// TwinCAT 3 PLC project TcForgeExample
// Title: TcForgeExample
// Company: Home
// ProjectVersion: 2.0.0.0
// ProgramVersion: 3.1.4026.26
// libraries:
//   Tc2_Standard, 3.4.7.0 (Beckhoff Automation GmbH)
//   Tc2_System, 3.10.2.0 (Beckhoff Automation GmbH)
//   Tc3_JsonXml, 3.4.9.0 (Beckhoff Automation GmbH)
//   Tc3_Module, 3.4.7.0 (Beckhoff Automation GmbH)
//   [TcForge], 2.0.0.0 (Home)
// project tree:
//   / PlcTask.TcTTO
//   Assembly/ GVL_HW.TcGVL, MAIN.TcPOU, FB_AssemblyStation.TcPOU, ST_AssemblyInputs.TcDUT, ST_AssemblyOutputs.TcDUT
//   ClampCycle/ FB_ReferenceMachine.TcPOU, E_ReferenceCommand.TcDUT
//   Simulation/ FB_SimulationBridge.TcPOU
//   Actuators/ FB_CylinderAssembly.TcPOU, ST_CylinderFeedback.TcDUT, ST_CylinderOutputs.TcDUT
//   Inspection/ FB_AssemblySensors.TcPOU
// (motion and I/O tree: see PLC project tcforge)
// real-time tasks:
//   TASK PlcTask: cycle T#10ms, priority 1, ADS port 350

CONFIGURATION TcForgeExample
    RESOURCE PLC ON TwinCAT3
        TASK PlcTask(INTERVAL := T#10ms, PRIORITY := 1);
        PROGRAM MAIN WITH PlcTask : MAIN;
    END_RESOURCE
END_CONFIGURATION

// ---- ClampCycle/E_ReferenceCommand.TcDUT
{attribute 'qualified_only'}
{attribute 'strict'}
TYPE E_ReferenceCommand : (None, Home, Start, Stop, Abort, Reset);
END_TYPE

// ---- Actuators/ST_CylinderFeedback.TcDUT
// Feedback belongs to the plant, not to the commanded direction.
TYPE ST_CylinderFeedback :
STRUCT
    advanced : BOOL;
    retracted : BOOL;
END_STRUCT
END_TYPE

// ---- Actuators/ST_CylinderOutputs.TcDUT
// Map these signals to the two valve coils at the application boundary.
TYPE ST_CylinderOutputs :
STRUCT
    advance : BOOL;
    retract : BOOL;
END_STRUCT
END_TYPE

// ---- Assembly/ST_AssemblyInputs.TcDUT
// Discrete assembly station: three cylinders and four measurement channels.
// The IO adapter supplies quality; default UNKNOWN deliberately inhibits motion.
TYPE ST_AssemblyInputs :
STRUCT
    clamp : ST_CylinderFeedback;
    press : ST_CylinderFeedback;
    ejector : ST_CylinderFeedback;

    partPresent : BOOL;       // Photoelectric sensor at the locating nest.
    dischargeClear : BOOL;    // Downstream sensor: permission to eject a part.
    pressureRaw : INT;        // 0..32767 maps to 0..10 bar.
    heightRaw : INT;          // 0..32767 maps to 0..20 mm.

    inputQuality : TcForge.E_IO_Quality := TcForge.E_IO_Quality.UNKNOWN;
    outputQuality : TcForge.E_IO_Quality := TcForge.E_IO_Quality.UNKNOWN;
    shutdownConfirmed : BOOL; // Independent plant feedback, never coil-derived.
    shutdownQuality : TcForge.E_IO_Quality := TcForge.E_IO_Quality.UNKNOWN;
END_STRUCT
END_TYPE

// ---- Assembly/ST_AssemblyOutputs.TcDUT
TYPE ST_AssemblyOutputs :
STRUCT
    clamp : ST_CylinderOutputs;
    press : ST_CylinderOutputs;
    ejector : ST_CylinderOutputs;
END_STRUCT
END_TYPE

// ---- Assembly/GVL_HW.TcGVL
// Application process image. Map physical terminals or a simulation adapter
// here, and derive quality from that adapter's actual communication health.
{attribute 'qualified_only'}
VAR_GLOBAL
    inputs : ST_AssemblyInputs;
    outputs : ST_AssemblyOutputs;
END_VAR

// ---- Assembly/MAIN.TcPOU
// Hardware mapping is kept here; the machine FB has no absolute IO addresses.
PROGRAM MAIN
VAR
    machine : FB_AssemblyStation;
    command : E_ReferenceCommand;
END_VAR

machine(inputs := GVL_HW.inputs, command := command);
GVL_HW.outputs := machine.outputs;

END_PROGRAM

// ---- Assembly/FB_AssemblyStation.TcPOU
// Machine recipe: locate -> press -> inspect -> release -> eject.
// Call once per scan. Devices never call the machine sequence themselves.
FUNCTION_BLOCK FB_AssemblyStation
VAR_INPUT
    inputs : ST_AssemblyInputs;
    command : E_ReferenceCommand; // Return to None before repeating a command.
    recoverOnOnlineChange : BOOL := TRUE; // Production-safe default; compatible edits may opt out.
END_VAR

VAR_OUTPUT
    outputs : ST_AssemblyOutputs;
    sequence : TcForge.ST_SM_Status;
    lastResponse : TcForge.E_RpcMethodResponse;
    outputsInhibited : BOOL;
    pressureBar : REAL;
    heightMm : REAL;
END_VAR

VAR
    // Physical areas: conditioning, locating nest, press and discharge.
    sensors : FB_AssemblySensors;
    clamp : FB_CylinderAssembly;
    press : FB_CylinderAssembly;
    ejector : FB_CylinderAssembly;

    // Machine lifecycle and execution ownership.
    sm : TcForge.FB_StateMachine;
    continuity : TcForge.FB_ExecutionContinuity;
    taskIndex : DINT;
    previousCommand : E_ReferenceCommand;
    freshCommand : BOOL;
    resetPending : BOOL;
    recoveryRequired : BOOL;
    healthy : BOOL;
    shutdownTrusted : BOOL;
    motionAllowed : BOOL;

    // One-scan direction requests. The actuator assembly handles coil policy.
    clampAdvance : BOOL;
    clampRetract : BOOL;
    pressAdvance : BOOL;
    pressRetract : BOOL;
    ejectAdvance : BOOL;
    ejectRetract : BOOL;

    // Each recipe phase owns a separate lifecycle instance.
    homePark : TcForge.FB_Step;
    homeUnclamp : TcForge.FB_Step;
    waitPart : TcForge.FB_Step;
    locatePart : TcForge.FB_Step;
    pressPart : TcForge.FB_Step;
    inspectPart : TcForge.FB_Step;
    withdrawPress : TcForge.FB_Step;
    releasePart : TcForge.FB_Step;
    ejectPart : TcForge.FB_Step;
    parkEjector : TcForge.FB_Step;
    stopStep : TcForge.FB_Step;
    abortStep : TcForge.FB_Step;
END_VAR

// 1. Detect interrupted execution before accepting any new command.
taskIndex := Tc2_System.GETCURTASKINDEXEX();
IF taskIndex > 0 THEN
    continuity(
        taskIndex := taskIndex,
        cycleCounter := TwinCAT_SystemInfoVarList._TaskInfo[taskIndex].CycleCount,
        onlineChangeCounter := TwinCAT_SystemInfoVarList._AppInfo.OnlineChangeCnt,
        recoverOnOnlineChange := recoverOnOnlineChange
    );
ELSE
    continuity(taskIndex := taskIndex);
END_IF;

IF continuity.interrupted THEN
    recoveryRequired := TRUE;
    sm.Abort();
END_IF;

// 2. Current input quality and air pressure gate every automatic movement.
sensors(inputs := inputs);
healthy := sensors.qualityGood AND sensors.pressureGood
    AND inputs.outputQuality = TcForge.E_IO_Quality.GOOD
    AND NOT (inputs.clamp.advanced AND inputs.clamp.retracted)
    AND NOT (inputs.press.advanced AND inputs.press.retracted)
    AND NOT (inputs.ejector.advanced AND inputs.ejector.retracted);
shutdownTrusted := inputs.shutdownConfirmed
    AND inputs.shutdownQuality = TcForge.E_IO_Quality.GOOD;

sm.cfgHome.nRequired := 1;
sm.cfgStart.nRequired := 1;
sm.cfgAuto.nRequired := 1;
sm.cfgRunning.nRequired := 1;
sm.MapHomeCondition(bitIndex := 0, bGood := healthy);
sm.MapStartCondition(bitIndex := 0, bGood := healthy);
sm.MapAutoCondition(bitIndex := 0, bGood := healthy);
sm.MapRunningIntlk(bitIndex := 0, bGood := healthy);

// 3. Commands are consumed once, including rejected commands.
resetPending := FALSE;
freshCommand := command <> E_ReferenceCommand.None AND command <> previousCommand;
previousCommand := command;
IF freshCommand THEN
    IF continuity.interrupted THEN
        lastResponse := TcForge.E_RpcMethodResponse.REJECTED_INTERLOCKED;
    ELSE
        HandleCommand();
    END_IF;
END_IF;

// Clear device faults and the recovered running-interlock latch before the
// state machine samples them. FB_Interlock publishes sts.bOK from its body, so
// resetting the latch after sm() would make this Reset fail for one scan.
IF resetPending THEN
    clamp.ResetFaults();
    press.ResetFaults();
    ejector.ResetFaults();
    sm.ResetRunningIntlk();
END_IF;

sm(
    inpSubmoduleFaulted := clamp.faulted OR press.faulted OR ejector.faulted,
    inpShutdownConfirmed := shutdownTrusted
);

// 4. Recipe methods only request moves; every device still executes below.
clampAdvance := FALSE;
clampRetract := FALSE;
pressAdvance := FALSE;
pressRetract := FALSE;
ejectAdvance := FALSE;
ejectRetract := FALSE;
RunHome();
RunCycle();
RunShutdown();

motionAllowed := healthy AND NOT recoveryRequired AND NOT sm.IsFaulted()
    AND NOT sm.Status.ShutdownFailed
    AND (sm.Status.State = TcForge.E_SM_State.HOMING
        OR sm.Status.State = TcForge.E_SM_State.RUNNING);

// 5. Geometry interlocks are checked at the actuator boundary every scan.
// The press cannot descend without the locating clamp; the ejector cannot
// enter the nest until the press and clamp are both retracted.
clamp(
    feedback := inputs.clamp,
    quality := inputs.inputQuality,
    outputQuality := inputs.outputQuality,
    permitMotion := motionAllowed,
    allowAdvance := inputs.press.retracted,
    allowRetract := inputs.press.retracted,
    requestAdvance := clampAdvance,
    requestRetract := clampRetract,
    requestReset := resetPending
);
press(
    feedback := inputs.press,
    quality := inputs.inputQuality,
    outputQuality := inputs.outputQuality,
    permitMotion := motionAllowed,
    allowAdvance := inputs.clamp.advanced AND sensors.partPresent,
    allowRetract := TRUE,
    requestAdvance := pressAdvance,
    requestRetract := pressRetract,
    requestReset := resetPending
);
ejector(
    feedback := inputs.ejector,
    quality := inputs.inputQuality,
    outputQuality := inputs.outputQuality,
    permitMotion := motionAllowed,
    allowAdvance := inputs.press.retracted AND inputs.clamp.retracted
        AND sensors.dischargeClear,
    allowRetract := TRUE,
    requestAdvance := ejectAdvance,
    requestRetract := ejectRetract,
    requestReset := resetPending
);

IF clamp.commandRejected OR press.commandRejected OR ejector.commandRejected THEN
    sm.Abort();
    recoveryRequired := TRUE;
END_IF;

IF resetPending THEN
    lastResponse := sm.Reset();
    IF lastResponse = TcForge.E_RpcMethodResponse.ACCEPTED THEN
        recoveryRequired := FALSE;
    END_IF;
END_IF;

// 6. Final process-image gate catches faults detected during this scan.
outputsInhibited := NOT motionAllowed OR clamp.faulted OR press.faulted
    OR ejector.faulted OR sm.IsFaulted() OR recoveryRequired;
outputs.clamp := clamp.outputs;
outputs.press := press.outputs;
outputs.ejector := ejector.outputs;
IF outputsInhibited THEN
    outputs.clamp.advance := FALSE;
    outputs.clamp.retract := FALSE;
    outputs.press.advance := FALSE;
    outputs.press.retract := FALSE;
    outputs.ejector.advance := FALSE;
    outputs.ejector.retract := FALSE;
END_IF;

sequence := sm.Status;
pressureBar := sensors.pressureBar;
heightMm := sensors.heightMm;

METHOD PRIVATE HandleCommand
CASE command OF
E_ReferenceCommand.Home:
    IF healthy AND NOT recoveryRequired THEN
        lastResponse := sm.Home();
    ELSE
        lastResponse := TcForge.E_RpcMethodResponse.REJECTED_INTERLOCKED;
    END_IF;

E_ReferenceCommand.Start:
    IF healthy AND NOT recoveryRequired THEN
        lastResponse := sm.Start();
    ELSE
        lastResponse := TcForge.E_RpcMethodResponse.REJECTED_INTERLOCKED;
    END_IF;

E_ReferenceCommand.Stop:
    lastResponse := sm.Stop();

E_ReferenceCommand.Abort:
    lastResponse := sm.Abort();

E_ReferenceCommand.Reset:
    IF sm.Status.State <> TcForge.E_SM_State.STOPPED THEN
        lastResponse := TcForge.E_RpcMethodResponse.REJECTED_WRONG_STATE;
    ELSIF NOT healthy OR NOT shutdownTrusted THEN
        lastResponse := TcForge.E_RpcMethodResponse.REJECTED_INTERLOCKED;
    ELSE
        resetPending := TRUE;
    END_IF;

ELSE
    lastResponse := TcForge.E_RpcMethodResponse.REJECTED_INVALID_PARAMETER;
END_CASE;
END_METHOD

METHOD PRIVATE RunHome
// 1000: Park press and ejector.
homePark(
    sm := sm,
    nStep := 1000,
    nNextStep := 1002,
    nRequired := 1,
    nTimeout := 10,
    sName := 'Park press and ejector'
);
IF homePark.Entry THEN
    pressRetract := TRUE;
    ejectRetract := TRUE;
END_IF;
IF homePark.Execute THEN
    homePark.MapPerm(
        nIndex := 0,
        sDescription := 'Park press and ejector',
        bValue := inputs.press.retracted AND inputs.ejector.retracted
    );
END_IF;

// 1002: Open locating clamp.
homeUnclamp(
    sm := sm,
    nStep := 1002,
    nNextStep := 0,
    nRequired := 1,
    nTimeout := 10,
    sName := 'Open locating clamp'
);
IF homeUnclamp.Entry THEN
    clampRetract := TRUE;
END_IF;
IF homeUnclamp.Execute THEN
    homeUnclamp.MapPerm(
        nIndex := 0,
        sDescription := 'Open locating clamp',
        bValue := inputs.clamp.retracted
    );
END_IF;
END_METHOD

METHOD PRIVATE RunCycle
// 3000: Wait for part in nest.
waitPart(
    sm := sm,
    nStep := 3000,
    nNextStep := 3002,
    nRequired := 1,
    nTimeout := 10,
    sName := 'Wait for part in nest'
);
IF waitPart.Execute THEN
    waitPart.MapPerm(
        nIndex := 0,
        sDescription := 'Wait for part in nest',
        bValue := sensors.partPresent
    );
END_IF;

// 3002: Locate part with clamp.
locatePart(
    sm := sm,
    nStep := 3002,
    nNextStep := 3004,
    nRequired := 1,
    nTimeout := 10,
    sName := 'Locate part with clamp'
);
IF locatePart.Entry THEN
    clampAdvance := TRUE;
END_IF;
IF locatePart.Execute THEN
    locatePart.MapPerm(
        nIndex := 0,
        sDescription := 'Locate part with clamp',
        bValue := inputs.clamp.advanced
    );
END_IF;

// 3004: Press assembly.
pressPart(
    sm := sm,
    nStep := 3004,
    nNextStep := 3006,
    nRequired := 1,
    nTimeout := 10,
    sName := 'Press assembly'
);
IF pressPart.Entry THEN
    pressAdvance := TRUE;
END_IF;
IF pressPart.Execute THEN
    pressPart.MapPerm(
        nIndex := 0,
        sDescription := 'Press assembly',
        bValue := inputs.press.advanced
    );
END_IF;

// 3006: Verify assembly height.
inspectPart(
    sm := sm,
    nStep := 3006,
    nNextStep := 3008,
    nRequired := 1,
    nTimeout := 10,
    sName := 'Verify assembly height'
);
IF inspectPart.Execute THEN
    inspectPart.MapPerm(
        nIndex := 0,
        sDescription := 'Verify assembly height',
        bValue := sensors.heightAccepted
    );
END_IF;

// 3008: Withdraw press.
withdrawPress(
    sm := sm,
    nStep := 3008,
    nNextStep := 3010,
    nRequired := 1,
    nTimeout := 10,
    sName := 'Withdraw press'
);
IF withdrawPress.Entry THEN
    pressRetract := TRUE;
END_IF;
IF withdrawPress.Execute THEN
    withdrawPress.MapPerm(
        nIndex := 0,
        sDescription := 'Withdraw press',
        bValue := inputs.press.retracted
    );
END_IF;

// 3010: Release locating clamp.
releasePart(
    sm := sm,
    nStep := 3010,
    nNextStep := 3012,
    nRequired := 1,
    nTimeout := 10,
    sName := 'Release locating clamp'
);
IF releasePart.Entry THEN
    clampRetract := TRUE;
END_IF;
IF releasePart.Execute THEN
    releasePart.MapPerm(
        nIndex := 0,
        sDescription := 'Release locating clamp',
        bValue := inputs.clamp.retracted
    );
END_IF;

// 3012: Eject finished part.
ejectPart(
    sm := sm,
    nStep := 3012,
    nNextStep := 3014,
    nRequired := 1,
    nTimeout := 10,
    sName := 'Eject finished part'
);
IF ejectPart.Entry THEN
    ejectAdvance := TRUE;
END_IF;
IF ejectPart.Execute THEN
    ejectPart.MapPerm(
        nIndex := 0,
        sDescription := 'Eject finished part',
        bValue := inputs.ejector.advanced AND NOT sensors.partPresent
    );
END_IF;

// 3014: Park ejector.
parkEjector(
    sm := sm,
    nStep := 3014,
    nNextStep := 0,
    nRequired := 1,
    nTimeout := 10,
    sName := 'Park ejector'
);
IF parkEjector.Entry THEN
    ejectRetract := TRUE;
END_IF;
IF parkEjector.Execute THEN
    parkEjector.MapPerm(
        nIndex := 0,
        sDescription := 'Park ejector',
        bValue := inputs.ejector.retracted
    );
END_IF;
END_METHOD

METHOD PRIVATE RunShutdown
// Stop and Abort remove all coil requests. Physical shutdown still requires
// independent feedback. Neither path guesses that an unpowered cylinder is home.
stopStep(
    sm := sm,
    nStep := 2000,
    nNextStep := 0,
    nRequired := 1,
    nTimeout := 5,
    sName := 'Confirm stopped station'
);
IF stopStep.Execute THEN
    stopStep.MapPerm(
        nIndex := 0,
        sDescription := 'Independent shutdown confirmed',
        bValue := shutdownTrusted
    );
END_IF;

abortStep(
    sm := sm,
    nStep := 5000,
    nNextStep := 0,
    nRequired := 1,
    nTimeout := 5,
    sName := 'Confirm aborted station'
);
IF abortStep.Execute THEN
    abortStep.MapPerm(
        nIndex := 0,
        sDescription := 'Independent shutdown confirmed',
        bValue := shutdownTrusted
    );
END_IF;
END_METHOD

END_FUNCTION_BLOCK

// ---- Inspection/FB_AssemblySensors.TcPOU
// Condition photoelectric and analog signals once per scan.
// The station consumes engineering units and quality, not raw terminal values.
FUNCTION_BLOCK FB_AssemblySensors
VAR_INPUT
    inputs : ST_AssemblyInputs;
END_VAR

VAR_OUTPUT
    partPresent : BOOL;
    dischargeClear : BOOL;
    pressureBar : REAL;
    heightMm : REAL;
    qualityGood : BOOL;
    pressureGood : BOOL;
    heightAccepted : BOOL;
END_VAR

VAR
    partSensor : TcForge.FB_DigitalInput;
    dischargeSensor : TcForge.FB_DigitalInput;
    pressureSensor : TcForge.FB_AnalogInput;
    heightSensor : TcForge.FB_AnalogInput;
    pressureValue : TcForge.U_IoRaw_In;
    heightValue : TcForge.U_IoRaw_In;
END_VAR

// Fixed example commissioning values. Production settings belong in a recipe
// or validated configuration; these values demonstrate engineering-unit scaling.
pressureSensor.cfg.euMax := 10.0;
pressureSensor.cfg.unit := TcForge.E_Unit.BAR;
heightSensor.cfg.euMax := 20.0;
heightSensor.cfg.unit := TcForge.E_Unit.MILLIMETER;
pressureValue.nInt := inputs.pressureRaw;
heightValue.nInt := inputs.heightRaw;

partSensor(inSignal := inputs.partPresent, inpQuality := inputs.inputQuality);
dischargeSensor(inSignal := inputs.dischargeClear, inpQuality := inputs.inputQuality);
pressureSensor(inRaw := pressureValue, inpQuality := inputs.inputQuality);
heightSensor(inRaw := heightValue, inpQuality := inputs.inputQuality);

partPresent := partSensor.sts.value;
dischargeClear := dischargeSensor.sts.value;
pressureBar := pressureSensor.sts.value;
heightMm := heightSensor.sts.value;

qualityGood := partSensor.sts.quality = TcForge.E_IO_Quality.GOOD
    AND dischargeSensor.sts.quality = TcForge.E_IO_Quality.GOOD
    AND pressureSensor.sts.quality = TcForge.E_IO_Quality.GOOD
    AND heightSensor.sts.quality = TcForge.E_IO_Quality.GOOD;

// Do not interpret a held measurement as fresh evidence after quality loss.
pressureGood := qualityGood AND pressureBar >= 5.0 AND pressureBar <= 8.0;
heightAccepted := qualityGood AND heightMm >= 9.5 AND heightMm <= 10.5;

END_FUNCTION_BLOCK

// ---- Actuators/FB_CylinderAssembly.TcPOU
// Reused by the locating clamp, press and ejector.
// Composes actuator supervision and both output policies in one owning task.
// Request inputs are one-scan pulses supplied by the station sequence.
FUNCTION_BLOCK FB_CylinderAssembly
VAR_INPUT
    feedback : ST_CylinderFeedback;
    quality : TcForge.E_IO_Quality := TcForge.E_IO_Quality.UNKNOWN;
    outputQuality : TcForge.E_IO_Quality := TcForge.E_IO_Quality.UNKNOWN;
    permitMotion : BOOL;
    allowAdvance : BOOL := TRUE;
    allowRetract : BOOL := TRUE;
    requestAdvance : BOOL;
    requestRetract : BOOL;
    requestReset : BOOL;
END_VAR

VAR_OUTPUT
    outputs : ST_CylinderOutputs;
    status : TcForge.ST_TwoPosActuator_Sts;
    faulted : BOOL;
    commandRejected : BOOL;
    lastResponse : TcForge.E_RpcMethodResponse;
END_VAR

VAR
    cylinder : TcForge.FB_TwoPosActuator;
    advanceCoil : TcForge.FB_DigitalOutput;
    retractCoil : TcForge.FB_DigitalOutput;
    feedbackGood : BOOL;
    motionAllowed : BOOL;
END_VAR

// 1. Evaluate this scan's feedback before admitting motion.
feedbackGood := quality = TcForge.E_IO_Quality.GOOD
    AND outputQuality = TcForge.E_IO_Quality.GOOD
    AND NOT (feedback.advanced AND feedback.retracted);

// Keep geometry/quality permissives evaluated while idle. The station motion
// gate is checked separately below, so a Home entry does not borrow a stale
// FALSE permission from the preceding STOPPED scan.
cylinder.cfgAdvancePermissives.nRequired := 1;
cylinder.cfgRetractPermissives.nRequired := 1;
cylinder.MapAdvanceCondition(bitIndex := 0, bGood := feedbackGood AND allowAdvance);
cylinder.MapRetractCondition(bitIndex := 0, bGood := feedbackGood AND allowRetract);

// Reset is a separate stationary operation; it cannot admit a simultaneous move.
commandRejected := FALSE;
IF requestReset AND feedbackGood THEN
    cylinder.Reset();
    advanceCoil.Reset();
    retractCoil.Reset();
END_IF;

motionAllowed := feedbackGood AND permitMotion AND NOT requestReset;
IF NOT motionAllowed THEN
    cylinder.Abort();
END_IF;

// 2. Issue at most one direction command. Rejections are visible to the step.
IF requestAdvance OR requestRetract THEN
    IF NOT motionAllowed OR (requestAdvance AND requestRetract) THEN
        lastResponse := TcForge.E_RpcMethodResponse.REJECTED_INTERLOCKED;
    ELSIF requestAdvance THEN
        lastResponse := cylinder.Advance();
    ELSE
        lastResponse := cylinder.Retract();
    END_IF;

    commandRejected := lastResponse <> TcForge.E_RpcMethodResponse.ACCEPTED
        AND lastResponse <> TcForge.E_RpcMethodResponse.REJECTED_ALREADY_AT_TARGET;
END_IF;

cylinder(
    inAdvanced := feedback.advanced,
    inRetracted := feedback.retracted
);

// 3. Apply final output policy after the actuator has detected current faults.
motionAllowed := motionAllowed AND NOT cylinder.IsFaulted()
    AND NOT advanceCoil.IsFaulted() AND NOT retractCoil.IsFaulted();

IF motionAllowed THEN
    IF cylinder.outAdvance THEN
        advanceCoil.SetOn();
    ELSE
        advanceCoil.SetOff();
    END_IF;

    IF cylinder.outRetract THEN
        retractCoil.SetOn();
    ELSE
        retractCoil.SetOff();
    END_IF;
ELSE
    advanceCoil.ForceSafe();
    retractCoil.ForceSafe();
END_IF;

advanceCoil(inpQuality := outputQuality);
retractCoil(inpQuality := outputQuality);

outputs.advance := advanceCoil.outSignal;
outputs.retract := retractCoil.outSignal;
status := cylinder.sts;
faulted := cylinder.IsFaulted() OR advanceCoil.IsFaulted()
    OR retractCoil.IsFaulted();

// The station admits this operation only when stopped, with trusted shutdown.
METHOD PUBLIC ResetFaults
cylinder.Reset();
advanceCoil.Reset();
retractCoil.Reset();

// Publish the cleared submodule status before the station evaluates Reset.
faulted := cylinder.IsFaulted() OR advanceCoil.IsFaulted()
    OR retractCoil.IsFaulted();
END_METHOD

END_FUNCTION_BLOCK

// ---- ClampCycle/FB_ReferenceMachine.TcPOU
// Application composition. Call exactly once per scan from one owning task.
// No RPC entry points. command is sampled by this cyclic body on value changes.
FUNCTION_BLOCK FB_ReferenceMachine
VAR_INPUT
    // Explicit application policy for compatible engineering edits; gaps still cancel motion.
    recoverOnOnlineChange : BOOL := TRUE;
    command : E_ReferenceCommand;
    inAdvanced, inRetracted : BOOL;
    inputQuality : TcForge.E_IO_Quality := TcForge.E_IO_Quality.UNKNOWN;
    outputQuality : TcForge.E_IO_Quality := TcForge.E_IO_Quality.UNKNOWN;
    // Independent feedback from the application/plant, never synthesized from command bits.
    shutdownConfirmed : BOOL;
    shutdownQuality : TcForge.E_IO_Quality := TcForge.E_IO_Quality.UNKNOWN;
END_VAR

VAR_OUTPUT
    outAdvance, outRetract : BOOL;
    sequence : TcForge.ST_SM_Status;
    actuator : TcForge.ST_TwoPosActuator_Sts;
    faulted, qualityGood, outputsInhibited : BOOL;
    lastResponse : TcForge.E_RpcMethodResponse;
END_VAR
VAR
    continuity : TcForge.FB_ExecutionContinuity;
    taskIndex : DINT;
    recoveryRequired : BOOL;
    sm : TcForge.FB_StateMachine;
    clamp : TcForge.FB_TwoPosActuator;
    advanceOutput, retractOutput : TcForge.FB_DigitalOutput;
    homeStep, advanceStep, retractStep, stopCancelStep, stopRetractStep, abortStep : TcForge.FB_Step;
    previousCommand : E_ReferenceCommand;
    freshCommand, resetPending, confirmed, permitMotion : BOOL;
    response : TcForge.E_RpcMethodResponse;
END_VAR

// Execution interruption cancels intent before command admission or output evaluation.
taskIndex := Tc2_System.GETCURTASKINDEXEX();
IF taskIndex > 0 THEN
    continuity(
        taskIndex := taskIndex,
        cycleCounter := TwinCAT_SystemInfoVarList._TaskInfo[taskIndex].CycleCount,
        onlineChangeCounter := TwinCAT_SystemInfoVarList._AppInfo.OnlineChangeCnt,
        recoverOnOnlineChange := recoverOnOnlineChange
    );
ELSE
    continuity(taskIndex := taskIndex);
END_IF;
IF continuity.interrupted THEN
    recoveryRequired := TRUE;
    sm.Abort();
    clamp.Abort();
    advanceOutput.ForceSafe();
    retractOutput.ForceSafe();
END_IF;

// 1. Sample quality and configure/map required conditions before any command.
qualityGood := inputQuality = TcForge.E_IO_Quality.GOOD AND outputQuality = TcForge.E_IO_Quality.GOOD;
confirmed := shutdownConfirmed AND shutdownQuality = TcForge.E_IO_Quality.GOOD;
sm.cfgHome.nRequired := 1;
sm.cfgStart.nRequired := 1;
sm.cfgAuto.nRequired := 1;
sm.cfgRunning.nRequired := 1;
sm.MapHomeCondition(bitIndex := 0, bGood := qualityGood);
sm.MapStartCondition(bitIndex := 0, bGood := qualityGood);
sm.MapAutoCondition(bitIndex := 0, bGood := qualityGood);
sm.MapRunningIntlk(bitIndex := 0, bGood := qualityGood);
clamp.cfgAdvancePermissives.nRequired := 1;
clamp.cfgRetractPermissives.nRequired := 1;
clamp.MapAdvanceCondition(bitIndex := 0, bGood := qualityGood);
clamp.MapRetractCondition(bitIndex := 0, bGood := qualityGood);
resetPending := FALSE;
freshCommand := command <> E_ReferenceCommand.None AND command <> previousCommand;
previousCommand := command;

IF freshCommand AND continuity.interrupted THEN
    lastResponse := TcForge.E_RpcMethodResponse.REJECTED_INTERLOCKED;
END_IF;

// 2. Commands are consumed once. A held or rejected command cannot become latent work.
IF freshCommand AND NOT continuity.interrupted THEN
    CASE command OF
        E_ReferenceCommand.Home:
        IF qualityGood AND NOT recoveryRequired THEN
            lastResponse := sm.Home();
        ELSE
            lastResponse := TcForge.E_RpcMethodResponse.REJECTED_INTERLOCKED;
        END_IF;
        E_ReferenceCommand.Start:
        IF qualityGood AND NOT recoveryRequired THEN
            lastResponse := sm.Start();
        ELSE
            lastResponse := TcForge.E_RpcMethodResponse.REJECTED_INTERLOCKED;
        END_IF;
        E_ReferenceCommand.Stop: lastResponse := sm.Stop();
        E_ReferenceCommand.Abort: lastResponse := sm.Abort();
        E_ReferenceCommand.Reset:
        IF sm.Status.State <> TcForge.E_SM_State.STOPPED THEN
            lastResponse := TcForge.E_RpcMethodResponse.REJECTED_WRONG_STATE;
        ELSIF NOT qualityGood OR NOT confirmed OR (inAdvanced AND inRetracted) THEN
            lastResponse := TcForge.E_RpcMethodResponse.REJECTED_INTERLOCKED;
        ELSE
            clamp.Reset();
            advanceOutput.Reset();
            retractOutput.Reset();
            sm.ResetRunningIntlk();
            resetPending := TRUE;
        END_IF;
    ELSE
        lastResponse := TcForge.E_RpcMethodResponse.REJECTED_INVALID_PARAMETER;
    END_CASE;
END_IF;

// 3. State machine runs once, then every step once (including inactive steps).
sm(inpSubmoduleFaulted := clamp.IsFaulted() OR advanceOutput.IsFaulted() OR retractOutput.IsFaulted(),
    inpShutdownConfirmed := confirmed);
IF resetPending THEN
    lastResponse := sm.Reset();
    IF lastResponse = TcForge.E_RpcMethodResponse.ACCEPTED THEN
        recoveryRequired := FALSE;
    END_IF;
END_IF;

homeStep(sm := sm, nStep := 1000, nNextStep := 0, nRequired := 3, nTimeout := 6, sName := 'Retract clamp');
IF homeStep.Entry THEN
    response := clamp.Retract();
    IF response <> TcForge.E_RpcMethodResponse.ACCEPTED AND response <> TcForge.E_RpcMethodResponse.REJECTED_ALREADY_AT_TARGET THEN
        homeStep.RaiseFault(code := TcForge.E_SM_Fault.StepUserFault,
            reason := 'Clamp rejected motion command');
    END_IF;
END_IF;
IF homeStep.Execute THEN
    homeStep.MapPerm(nIndex := 0,
        sDescription := 'Position confirmed',
        bValue := inRetracted AND NOT inAdvanced);
    homeStep.MapPerm(nIndex := 1, sDescription := 'IO quality good', bValue := qualityGood);
END_IF;

advanceStep(sm := sm,
    nStep := 3000,
    nNextStep := 3002,
    nRequired := 3,
    nTimeout := 6,
    sName := 'Advance clamp');
IF advanceStep.Entry THEN
    response := clamp.Advance();
    IF response <> TcForge.E_RpcMethodResponse.ACCEPTED AND response <> TcForge.E_RpcMethodResponse.REJECTED_ALREADY_AT_TARGET THEN
        advanceStep.RaiseFault(code := TcForge.E_SM_Fault.StepUserFault,
            reason := 'Clamp rejected motion command');
    END_IF;
END_IF;
IF advanceStep.Execute THEN
    advanceStep.MapPerm(nIndex := 0,
        sDescription := 'Position confirmed',
        bValue := inAdvanced AND NOT inRetracted);
    advanceStep.MapPerm(nIndex := 1, sDescription := 'IO quality good', bValue := qualityGood);
END_IF;

retractStep(sm := sm, nStep := 3002, nNextStep := 0, nRequired := 3, nTimeout := 6, sName := 'Retract clamp');
IF retractStep.Entry THEN
    response := clamp.Retract();
    IF response <> TcForge.E_RpcMethodResponse.ACCEPTED AND response <> TcForge.E_RpcMethodResponse.REJECTED_ALREADY_AT_TARGET THEN
        retractStep.RaiseFault(code := TcForge.E_SM_Fault.StepUserFault,
            reason := 'Clamp rejected motion command');
    END_IF;
END_IF;
IF retractStep.Execute THEN
    retractStep.MapPerm(nIndex := 0,
        sDescription := 'Position confirmed',
        bValue := inRetracted AND NOT inAdvanced);
    retractStep.MapPerm(nIndex := 1, sDescription := 'IO quality good', bValue := qualityGood);
END_IF;

stopRetractStep(sm := sm,
    nStep := 2002,
    nNextStep := 0,
    nRequired := 3,
    nTimeout := 6,
    sName := 'Retract clamp');
IF stopRetractStep.Entry THEN
    response := clamp.Retract();
    IF response <> TcForge.E_RpcMethodResponse.ACCEPTED AND response <> TcForge.E_RpcMethodResponse.REJECTED_ALREADY_AT_TARGET THEN
        stopRetractStep.RaiseFault(code := TcForge.E_SM_Fault.StepUserFault,
            reason := 'Clamp rejected motion command');
    END_IF;
END_IF;
IF stopRetractStep.Execute THEN
    stopRetractStep.MapPerm(nIndex := 0,
        sDescription := 'Position confirmed',
        bValue := inRetracted AND NOT inAdvanced);
    stopRetractStep.MapPerm(nIndex := 1, sDescription := 'IO quality good', bValue := qualityGood);
END_IF;

stopCancelStep(sm := sm,
    nStep := 2000,
    nNextStep := 2002,
    nRequired := 0,
    nTimeout := 2,
    sName := 'Cancel motion before retract');
IF stopCancelStep.Entry THEN
    clamp.Abort();
END_IF;
abortStep(sm := sm,
    nStep := 5000,
    nNextStep := 0,
    nRequired := 1,
    nTimeout := 2,
    sName := 'Confirm shutdown');
IF abortStep.Entry THEN
    clamp.Abort();
END_IF;
IF abortStep.Execute THEN
    abortStep.MapPerm(nIndex := 0, sDescription := 'Independent shutdown feedback', bValue := confirmed);
END_IF;

// 4. Monitor the actuator with this scan's feedback and permissives.
// Inhibition also cancels internal motion so stale intent cannot reappear later.
permitMotion := qualityGood AND NOT recoveryRequired AND NOT sm.IsFaulted() AND NOT sm.Status.ShutdownFailed AND
(sm.Status.State = TcForge.E_SM_State.HOMING OR sm.Status.State = TcForge.E_SM_State.RUNNING OR sm.Status.State = TcForge.E_SM_State.STOPPING);
IF NOT permitMotion THEN
    clamp.Abort();
END_IF;
clamp(inAdvanced := inAdvanced, inRetracted := inRetracted);

// 5. Final output policy runs AFTER all fault detection and lifecycle commands.
permitMotion := permitMotion AND NOT clamp.IsFaulted() AND NOT advanceOutput.IsFaulted() AND NOT retractOutput.IsFaulted();
IF permitMotion THEN
    IF clamp.outAdvance THEN
        advanceOutput.SetOn();
    ELSE
        advanceOutput.SetOff();
    END_IF;
    IF clamp.outRetract THEN
        retractOutput.SetOn();
    ELSE
        retractOutput.SetOff();
    END_IF;
ELSE
    advanceOutput.ForceSafe();
    retractOutput.ForceSafe();
END_IF;
advanceOutput(inpQuality := outputQuality);
retractOutput(inpQuality := outputQuality);
outAdvance := advanceOutput.outSignal;
outRetract := retractOutput.outSignal;
outputsInhibited := NOT permitMotion;
faulted := sm.IsFaulted() OR clamp.IsFaulted() OR advanceOutput.IsFaulted() OR retractOutput.IsFaulted();
sequence := sm.Status;
actuator := clamp.sts;

END_FUNCTION_BLOCK

// ---- Simulation/FB_SimulationBridge.TcPOU
// PLC-owned exchange boundary for the complete discrete assembly station.
// Python supplies one coherent plant-input frame; this cyclic owner alone runs
// the controller and publishes its six output coils.
FUNCTION_BLOCK FB_SimulationBridge
VAR_INPUT
    recoverOnOnlineChange : BOOL := TRUE;
END_VAR

VAR_OUTPUT
    outClampAdvance, outClampRetract : BOOL;
    outPressAdvance, outPressRetract : BOOL;
    outEjectorAdvance, outEjectorRetract : BOOL;
END_VAR

VAR
    continuity : TcForge.FB_ExecutionContinuity;
    machine : FB_AssemblyStation;
    stationInputs : ST_AssemblyInputs;
    mutex : BOOL;
    boot, cycle, session, submitted, applied, lastAck : ULINT;
    pending, hasFrame, freshPrevious, newClaim : BOOL;
    pendingClampAdvanced, pendingClampRetracted : BOOL;
    pendingPressAdvanced, pendingPressRetracted : BOOL;
    pendingEjectorAdvanced, pendingEjectorRetracted : BOOL;
    pendingPartPresent, pendingDischargeClear : BOOL;
    pendingShutdown, pendingQuality : BOOL;
    pendingPressureRaw, pendingHeightRaw : INT;
    pendingCommand : UINT;
    command : E_ReferenceCommand;
    quality : TcForge.E_IO_Quality;
    watchdog : TON;
    owner : DINT;
    ownershipConflict : BOOL;
END_VAR

// 1. Serialize RPC exchange state with the owning PLC task.
IF NOT Tc2_System.TestAndSet(mutex) THEN
    RETURN;
END_IF;
IF owner = 0 THEN
    owner := Tc2_System.GETCURTASKINDEXEX();
    IF owner <= 0 THEN
        owner := 0;
        mutex := FALSE;
        RETURN;
    END_IF;
    boot := Tc2_System.F_GetSystemTime();
END_IF;
IF Tc2_System.GETCURTASKINDEXEX() <> owner THEN
    ownershipConflict := TRUE;
    session := 0;
    pending := FALSE;
    hasFrame := FALSE;
    outClampAdvance := FALSE;
    outClampRetract := FALSE;
    outPressAdvance := FALSE;
    outPressRetract := FALSE;
    outEjectorAdvance := FALSE;
    outEjectorRetract := FALSE;
    mutex := FALSE;
    RETURN;
END_IF;

// 2. Any execution gap rotates the epoch and discards unconsumed input.
continuity(
    taskIndex := owner,
    cycleCounter := TwinCAT_SystemInfoVarList._TaskInfo[owner].CycleCount,
    onlineChangeCounter := TwinCAT_SystemInfoVarList._AppInfo.OnlineChangeCnt,
    recoverOnOnlineChange := recoverOnOnlineChange
);
IF continuity.interrupted THEN
    boot := Tc2_System.F_GetSystemTime();
    session := 0;
    pending := FALSE;
    hasFrame := FALSE;
    freshPrevious := FALSE;
    newClaim := FALSE;
    submitted := 0;
    applied := 0;
    lastAck := 0;
    pendingCommand := 0;
    watchdog(IN := FALSE, PT := T#250MS);
END_IF;

// 3. Expire stale writers independently of the Python process.
watchdog(IN := session <> 0 AND NOT freshPrevious, PT := T#250MS);
freshPrevious := FALSE;
IF newClaim THEN
    watchdog(IN := FALSE, PT := T#250MS);
    newClaim := FALSE;
END_IF;
IF watchdog.Q OR ownershipConflict THEN
    session := 0;
    pending := FALSE;
    hasFrame := FALSE;
END_IF;

// 4. Apply an admitted frame atomically at the scan boundary.
command := E_ReferenceCommand.None;
IF pending AND session <> 0 THEN
    stationInputs.clamp.advanced := pendingClampAdvanced;
    stationInputs.clamp.retracted := pendingClampRetracted;
    stationInputs.press.advanced := pendingPressAdvanced;
    stationInputs.press.retracted := pendingPressRetracted;
    stationInputs.ejector.advanced := pendingEjectorAdvanced;
    stationInputs.ejector.retracted := pendingEjectorRetracted;
    stationInputs.partPresent := pendingPartPresent;
    stationInputs.dischargeClear := pendingDischargeClear;
    stationInputs.pressureRaw := pendingPressureRaw;
    stationInputs.heightRaw := pendingHeightRaw;
    stationInputs.shutdownConfirmed := pendingShutdown;
    CASE pendingCommand OF
        1: command := E_ReferenceCommand.Home;
        2: command := E_ReferenceCommand.Start;
        3: command := E_ReferenceCommand.Stop;
        4: command := E_ReferenceCommand.Abort;
        5: command := E_ReferenceCommand.Reset;
    END_CASE;
    applied := submitted;
    pending := FALSE;
    hasFrame := TRUE;
    freshPrevious := TRUE;
END_IF;

IF hasFrame AND session <> 0 AND pendingQuality AND NOT ownershipConflict THEN
    quality := TcForge.E_IO_Quality.GOOD;
ELSE
    quality := TcForge.E_IO_Quality.BAD;
END_IF;
stationInputs.inputQuality := quality;
stationInputs.outputQuality := quality;
stationInputs.shutdownQuality := quality;

// 5. The production-style controller runs every available PLC scan.
machine(
    inputs := stationInputs,
    command := command,
    recoverOnOnlineChange := recoverOnOnlineChange
);
outClampAdvance := machine.outputs.clamp.advance AND quality = TcForge.E_IO_Quality.GOOD;
outClampRetract := machine.outputs.clamp.retract AND quality = TcForge.E_IO_Quality.GOOD;
outPressAdvance := machine.outputs.press.advance AND quality = TcForge.E_IO_Quality.GOOD;
outPressRetract := machine.outputs.press.retract AND quality = TcForge.E_IO_Quality.GOOD;
outEjectorAdvance := machine.outputs.ejector.advance AND quality = TcForge.E_IO_Quality.GOOD;
outEjectorRetract := machine.outputs.ejector.retract AND quality = TcForge.E_IO_Quality.GOOD;
cycle := cycle + 1;
mutex := FALSE;

{attribute 'TcRpcEnable' := '1'}
METHOD PUBLIC Identity : STRING(80)
Identity := 'TcForge.DiscreteAssembly/2';
END_METHOD

{attribute 'TcRpcEnable' := '1'}
METHOD PUBLIC Claim : DINT
VAR_INPUT
    client : ULINT;
    expectedBoot : ULINT;
END_VAR
Claim := 30;
IF client = 0 THEN RETURN; END_IF;
Claim := 22;
IF NOT Tc2_System.TestAndSet(mutex) THEN RETURN; END_IF;
IF boot = 0 OR owner = 0 THEN
    Claim := 12;
ELSIF ownershipConflict THEN
    Claim := 13;
ELSIF expectedBoot <> boot THEN
    Claim := 34;
ELSIF session <> 0 THEN
    IF client = session THEN Claim := 0; ELSE Claim := 11; END_IF;
ELSE
    session := client;
    submitted := 0;
    applied := 0;
    lastAck := 0;
    pending := FALSE;
    hasFrame := FALSE;
    newClaim := TRUE;
    Claim := 0;
END_IF;
mutex := FALSE;
END_METHOD

{attribute 'TcRpcEnable' := '1'}
METHOD PUBLIC Exchange : DINT
VAR_INPUT
    client, expectedBoot, frame, outputFrame : ULINT;
    clampAdvanced, clampRetracted : BOOL;
    pressAdvanced, pressRetracted : BOOL;
    ejectorAdvanced, ejectorRetracted : BOOL;
    partPresent, dischargeClear : BOOL;
    pressureRaw, heightRaw : INT;
    shutdownConfirmed, qualityGood : BOOL;
    requestedCommand : UINT;
END_VAR
Exchange := 30;
IF client = 0 OR frame = 0 OR requestedCommand > 5 THEN RETURN; END_IF;
Exchange := 22;
IF NOT Tc2_System.TestAndSet(mutex) THEN RETURN; END_IF;
IF expectedBoot <> boot THEN
    Exchange := 34;
ELSIF session = 0 OR watchdog.Q THEN
    Exchange := 12;
ELSIF client <> session THEN
    Exchange := 11;
ELSIF frame <= submitted THEN
    Exchange := 35;
ELSIF frame <> submitted + 1 OR outputFrame <= lastAck OR outputFrame > cycle THEN
    Exchange := 30;
ELSIF NOT pending THEN
    pendingClampAdvanced := clampAdvanced;
    pendingClampRetracted := clampRetracted;
    pendingPressAdvanced := pressAdvanced;
    pendingPressRetracted := pressRetracted;
    pendingEjectorAdvanced := ejectorAdvanced;
    pendingEjectorRetracted := ejectorRetracted;
    pendingPartPresent := partPresent;
    pendingDischargeClear := dischargeClear;
    pendingPressureRaw := pressureRaw;
    pendingHeightRaw := heightRaw;
    pendingShutdown := shutdownConfirmed;
    pendingQuality := qualityGood;
    pendingCommand := requestedCommand;
    submitted := frame;
    lastAck := outputFrame;
    pending := TRUE;
    Exchange := 1;
END_IF;
mutex := FALSE;
END_METHOD

{attribute 'TcRpcEnable' := '1'}
METHOD PUBLIC Release : DINT
VAR_INPUT
    client, expectedBoot : ULINT;
END_VAR
Release := 22;
IF NOT Tc2_System.TestAndSet(mutex) THEN RETURN; END_IF;
IF expectedBoot <> boot THEN
    Release := 34;
ELSIF session = 0 OR client <> session THEN
    Release := 11;
ELSE
    session := 0;
    hasFrame := FALSE;
    pending := FALSE;
    Release := 0;
END_IF;
mutex := FALSE;
END_METHOD

{attribute 'TcRpcEnable' := '1'}
METHOD PUBLIC Snapshot : STRING(255)
Snapshot := '22';
IF NOT Tc2_System.TestAndSet(mutex) THEN RETURN; END_IF;
Snapshot := '0';
Snapshot := CONCAT(Snapshot, CONCAT(',', ULINT_TO_STRING(boot)));
Snapshot := CONCAT(Snapshot, CONCAT(',', ULINT_TO_STRING(cycle)));
Snapshot := CONCAT(Snapshot, CONCAT(',', ULINT_TO_STRING(applied)));
Snapshot := CONCAT(Snapshot, CONCAT(',', DINT_TO_STRING(BOOL_TO_UINT(outClampAdvance))));
Snapshot := CONCAT(Snapshot, CONCAT(',', DINT_TO_STRING(BOOL_TO_UINT(outClampRetract))));
Snapshot := CONCAT(Snapshot, CONCAT(',', DINT_TO_STRING(BOOL_TO_UINT(outPressAdvance))));
Snapshot := CONCAT(Snapshot, CONCAT(',', DINT_TO_STRING(BOOL_TO_UINT(outPressRetract))));
Snapshot := CONCAT(Snapshot, CONCAT(',', DINT_TO_STRING(BOOL_TO_UINT(outEjectorAdvance))));
Snapshot := CONCAT(Snapshot, CONCAT(',', DINT_TO_STRING(BOOL_TO_UINT(outEjectorRetract))));
Snapshot := CONCAT(Snapshot, CONCAT(',', DINT_TO_STRING(machine.sequence.State)));
Snapshot := CONCAT(Snapshot, CONCAT(',', DINT_TO_STRING(BOOL_TO_UINT(machine.sequence.Faulted))));
Snapshot := CONCAT(Snapshot, CONCAT(',', DINT_TO_STRING(BOOL_TO_UINT(machine.outputsInhibited))));
Snapshot := CONCAT(Snapshot, CONCAT(',', DINT_TO_STRING(machine.lastResponse)));
Snapshot := CONCAT(Snapshot, CONCAT(',', ULINT_TO_STRING(session)));
Snapshot := CONCAT(Snapshot, CONCAT(',', DINT_TO_STRING(owner)));
Snapshot := CONCAT(Snapshot, CONCAT(',', DINT_TO_STRING(BOOL_TO_UINT(quality = TcForge.E_IO_Quality.GOOD AND NOT watchdog.Q))));
Snapshot := CONCAT(Snapshot, CONCAT(',', DINT_TO_STRING(machine.sequence.Step.Current)));
mutex := FALSE;
END_METHOD

END_FUNCTION_BLOCK
